(* IEC 61131-3 sources: Temperature-Cabinet-Control-Automation/src/POUs, 3 files *)

(* ---- FB_CabinetSetpointControl.st ---- *)
(*
    FUNCTION_BLOCK: FB_CabinetSetpointControl
    Project:  Temperature Cabinet Setpoint Control from CODESYS HMI
    Author:   OJ (Omkar Joshi) - Oliver Mechatronics
    Language: IEC 61131-3 Structured Text (CODESYS 3.5, WebVisu)

    ------------------------------------------------------------------
    ROLE
    Supervisory setpoint control for the Left Hand Small Temperature
    Cabinet (Watlow F4S, Modbus RTU / RS-232). CODESYS never runs the
    thermal loop - the F4S keeps its own closed-loop PID. This block:

      1. Takes a new desired setpoint from the HMI (GVL_HMI.rReqSetpoint).
      2. Validates it against safe limits.
      3. Writes it once (edge-triggered FC06) to register 300 (SP1).
      4. Confirms acceptance by reading register 300 back and comparing.
      5. Raises a clear, prioritised fault if the write fails, the link
         is lost, the value is refused, or the cabinet is over temperature.

    Matches the Project Development Package spec (Details A) and the
    build guide already in codesys-modbus-integration/README.md
    (Part 3, Part 4) and the T1-T9 test plan in the main README.

    SCALING
    F4S registers carry one implied decimal (raw 1300 == 130.0 degC).
    rScale defaults to 10.0; change it if the unit is reconfigured
    for a different resolution.

    NOTE (known follow-up item): this FB reads/writes GVL_Modbus and
    GVL_HMI directly in its body rather than exclusively through
    VAR_INPUT/VAR_OUTPUT. That is how the Project Development Package
    and the README build guide specify it, and it is what the T1-T9
    bench tests exercise - but it does mean this FB cannot be unit
    tested or reused against a second GVL_Modbus instance without
    editing the body. See PLC_PRG for the wired-up call, and note the
    xOverTempDI placeholder wiring there.
    ------------------------------------------------------------------
*)
FUNCTION_BLOCK FB_CabinetSetpointControl
VAR_INPUT
    rRequestedSetpoint  : REAL;                    (* deg C from HMI                    *)
    xSetCommand         : BOOL;                    (* HMI SET - rising edge applies      *)
    xReset              : BOOL;                    (* fault reset - rising edge clears   *)
    xOverTempDI         : BOOL;                    (* spare EL1409 DI, TRUE = over-temp  *)

    (* ---- configurable, default to confirmed values ---- *)
    rMinSetpoint        : REAL := -40.0;           (* Lower safe bound, degC              *)
    rMaxSetpoint        : REAL := 200.0;           (* Upper safe bound, degC              *)
    rScale              : REAL := 10.0;            (* eng <-> raw multiplier              *)
    rTolerance          : REAL := 0.1;             (* deg C read-back tolerance           *)
    tCommsTimeout       : TIME := T#3S;            (* watchdog                            *)
END_VAR
VAR_OUTPUT
    eState              : E_SetpointState;
    eFault              : E_FaultCode;
    xConfirmed          : BOOL;
    xFault              : BOOL;
    rActualTemp         : REAL;                    (* Live chamber temperature, degC      *)
    rConfirmedSetpoint  : REAL;                    (* Last accepted setpoint, degC        *)
END_VAR
VAR
    rtrigSet            : R_TRIG;                  (* Edge detect on SET command          *)
    rtrigReset          : R_TRIG;                  (* Edge detect on RESET command        *)
    tonWatchdog         : TON;                     (* Comms-loss debounce                 *)
    tonConfirmWait      : TON;                     (* Read-back confirm timeout           *)
    wTargetRaw          : WORD;                    (* Setpoint being written, raw x10     *)
    rReadBack           : REAL;                    (* Setpoint echo, engineering units    *)
END_VAR

(* ---- Edge detect ---- *)
rtrigSet(CLK := xSetCommand);
rtrigReset(CLK := xReset);

(* ---- Always-live scaling of the cyclic read ---- *)
rActualTemp          := WORD_TO_REAL(GVL_Modbus.wInput1Value) / rScale;
rReadBack             := WORD_TO_REAL(GVL_Modbus.wSetpoint1Read) / rScale;
GVL_HMI.rChamberTemp := rActualTemp;

(* ---- Comms watchdog: LEVEL signal, NOT an edge pulse (avoids R_TRIG->TON trap) ---- *)
tonWatchdog(IN := NOT GVL_Modbus.xModbusDone, PT := tCommsTimeout);

(* ---- Over-temp interlock (highest priority latch) ---- *)
IF xOverTempDI THEN
    eFault := E_FaultCode.OVER_TEMP;
    eState := E_SetpointState.FAULTED;
END_IF

(* ---- Comms loss latch (any state) ---- *)
IF tonWatchdog.Q OR GVL_Modbus.xModbusError THEN
    eFault := E_FaultCode.COMMS_TIMEOUT;
    eState := E_SetpointState.FAULTED;
END_IF

CASE eState OF

    E_SetpointState.IDLE:
        xConfirmed := TRUE;
        GVL_Modbus.xWriteTrigger := FALSE;
        IF rtrigSet.Q THEN
            eState := E_SetpointState.READY;
        END_IF

    E_SetpointState.READY:
        xConfirmed := FALSE;
        IF rRequestedSetpoint < rMinSetpoint THEN
            eFault := E_FaultCode.RANGE_LOW;
            eState := E_SetpointState.FAULTED;
        ELSIF rRequestedSetpoint > rMaxSetpoint THEN
            eFault := E_FaultCode.RANGE_HIGH;
            eState := E_SetpointState.FAULTED;
        ELSE
            wTargetRaw := REAL_TO_WORD(rRequestedSetpoint * rScale);
            GVL_Modbus.wSetpoint1Write := wTargetRaw;
            eState := E_SetpointState.WRITING;
        END_IF

    E_SetpointState.WRITING:
        GVL_Modbus.xWriteTrigger := TRUE;    (* one-shot rising edge fires FC06 *)
        eState := E_SetpointState.CONFIRM;

    E_SetpointState.CONFIRM:
        GVL_Modbus.xWriteTrigger := FALSE;   (* drop trigger to re-arm the edge *)
        tonConfirmWait(IN := TRUE, PT := tCommsTimeout);
        IF ABS(rReadBack - rRequestedSetpoint) <= rTolerance THEN
            rConfirmedSetpoint := rReadBack;
            GVL_HMI.rConfirmedSetpoint := rReadBack;
            tonConfirmWait(IN := FALSE);
            eState := E_SetpointState.IDLE;
        ELSIF tonConfirmWait.Q THEN
            eFault := E_FaultCode.NOT_ACCEPTED;
            eState := E_SetpointState.FAULTED;
        END_IF

    E_SetpointState.FAULTED:
        xConfirmed := FALSE;
        GVL_Modbus.xWriteTrigger := FALSE;
        (* Latched - clears only on reset edge AND only if condition is gone *)
        IF rtrigReset.Q
           AND NOT xOverTempDI
           AND NOT tonWatchdog.Q
           AND NOT GVL_Modbus.xModbusError THEN
            eFault := E_FaultCode.NO_FAULT;
            eState := E_SetpointState.IDLE;
        END_IF

END_CASE

xFault                      := (eState = E_SetpointState.FAULTED);
GVL_HMI.xSetpointConfirmed  := xConfirmed AND NOT xFault;
GVL_HMI.xFaultActive        := xFault;
GVL_HMI.eFaultCode          := eFault;

(* ---- PLC_PRG.st ---- *)
(*
    PROGRAM:  PLC_PRG
    Project:  Temperature Cabinet Setpoint Control from CODESYS HMI
    Author:   OJ (Omkar Joshi) - Oliver Mechatronics
    Language: IEC 61131-3 Structured Text (CODESYS 3.5, WebVisu)

    Cyclic entry point (MainTask). Instantiates the supervisory setpoint
    controller. Because FB_CabinetSetpointControl reads/writes GVL_Modbus
    and GVL_HMI directly in its body (see that FB's header note), this
    program only needs to pass through the operator-facing parameters
    and the safety interlock input.

    Matches the Project Development Package spec (Details A) and the
    build guide already in codesys-modbus-integration/README.md.

    TODO (flagged in the Project Development Package, not yet resolved):
    xOverTempDI below is wired to GVL_Modbus.xModbusError as a
    placeholder. REPLACE with the real mapped EL1409 digital-input
    channel (spare over-temperature lamp contact) in the EtherCAT I/O
    mapping before relying on this interlock.
*)
PROGRAM PLC_PRG
VAR
    fbSetpoint : FB_CabinetSetpointControl;
END_VAR

(* ---- Drive the supervisory setpoint controller ---- *)
fbSetpoint(
    rRequestedSetpoint := GVL_HMI.rReqSetpoint,
    xSetCommand        := GVL_HMI.xSetBtn,
    xReset             := GVL_HMI.xResetBtn,
    xOverTempDI        := GVL_Modbus.xModbusError,  (* REPLACE with mapped EL1409 DI channel *)
    rMinSetpoint       := 30.0,
    rMaxSetpoint       := 130.0
);

(* ---- Consume dialog button one-shots ---- *)
GVL_HMI.xSetBtn   := FALSE;
GVL_HMI.xResetBtn := FALSE;

(* ---- PLC_PRG_TCP_Retargeted.st ---- *)
PROGRAM PLC_PRG
(* ======================================================================
   Retargeted for TCP register sources (Python gateway via Modbus TCP)
   ======================================================================
   Serial device abandoned. All reads/writes now come via the TCP slave
   device on the Modbus TCP master branch of the device tree.

   Proven register map (TCP holding registers, x10 integers):
     reg2 = chamber temperature (read-only, cyclic)
     reg3 = confirmed setpoint read-back (read-only, cyclic)
     reg4 = status/fault code (read-only, cyclic)
     reg0 = requested setpoint (write, cyclic or rising)
     reg1 = apply trigger (write, rising edge)

   I/O Mapping binds these to GVL_Modbus:
     reg2 -> wInput1Value (temperature)
     reg3 -> wSetpoint1Read (confirmed SP)
     reg4 -> wStatus (fault code: 0=OK, 2=WRITE_FAILED, 3=NOT_ACCEPTED, 4=RANGE, 5=COMMS)
     reg0 -> wSetpoint1Write (requested SP, x10)
     reg1 -> xWriteTrigger (apply pulse, BOOL as WORD 0/1)

   The state machine logic is unchanged from the serial version. Only the
   data sources changed: TCP channels instead of serial channels.
   ====================================================================== *)

VAR
    rChamberTemp        : REAL;
    rReqSetpoint        : REAL := 26.5;           (* set in watch window or WebVisu *)
    rConfirmedSetpoint  : REAL;

    rMinSetpoint        : REAL := -40.0;
    rMaxSetpoint        : REAL := 200.0;

    eSetpointState      : E_SetpointState := E_SetpointState.IDLE;
    eFaultCode          : E_FaultCode := E_FaultCode.NO_FAULT;

    xStartWrite         : BOOL := FALSE;          (* rising-edge trigger for manual test *)
    xPrevStartWrite     : BOOL := FALSE;
    xWriteTriggered     : BOOL := FALSE;

    dwWriteTimeout      : DWORD := 0;
    dwMaxTimeout        : DWORD := 300;           (* ~3s at 10ms MainTask *)
END_VAR

(* --- STEP 1: Scale raw TCP values -> engineering units ---
   TCP registers carry x10 integers; we work in real degrees.
   All three reads come from the TCP channels (wInput1Value, wSetpoint1Read, wStatus).
*)
rChamberTemp       := GVL_Modbus.wInput1Value / 10.0;
rConfirmedSetpoint := GVL_Modbus.wSetpoint1Read / 10.0;

(* --- STEP 2: Detect rising edge on the manual test trigger ---
   When testing from watch window, toggle xStartWrite from FALSE to TRUE.
   In production (WebVisu or SCADA), the operator triggers via a button that
   sets a HMI variable, but the edge logic is the same.
*)
xWriteTriggered := (xStartWrite AND NOT xPrevStartWrite);
xPrevStartWrite := xStartWrite;

(* --- STEP 3: State machine (unchanged logic, TCP-based register sources) --- *)

CASE eSetpointState OF

    E_SetpointState.IDLE:
        (* Waiting for a write request. Hold the apply trigger low. *)
        GVL_Modbus.xWriteTrigger := FALSE;
        dwWriteTimeout := 0;

        IF xWriteTriggered THEN
            eSetpointState := E_SetpointState.READY;
        END_IF

    E_SetpointState.READY:
        (* Validate the requested setpoint against limits. *)
        IF rReqSetpoint < rMinSetpoint THEN
            eFaultCode := E_FaultCode.RANGE_LOW;
            eSetpointState := E_SetpointState.FAULTED;

        ELSIF rReqSetpoint > rMaxSetpoint THEN
            eFaultCode := E_FaultCode.RANGE_HIGH;
            eSetpointState := E_SetpointState.FAULTED;

        ELSE
            (* Valid range. Stage the request (x10 int) into the TCP write register. *)
            GVL_Modbus.wSetpoint1Write := DWORD_TO_WORD(REAL_TO_DWORD(rReqSetpoint * 10.0));
            eSetpointState := E_SetpointState.WRITING;
        END_IF

    E_SetpointState.WRITING:
        (* Pulse the apply trigger (one scan). The Python gateway services this
           by writing reg1=1 over RTU and then clearing it to 0 when done. *)
        GVL_Modbus.xWriteTrigger := TRUE;
        dwWriteTimeout := 0;
        eSetpointState := E_SetpointState.CONFIRM;

    E_SetpointState.CONFIRM:
        (* Drop the trigger immediately to re-arm the edge for the next request. *)
        GVL_Modbus.xWriteTrigger := FALSE;
        dwWriteTimeout := dwWriteTimeout + 1;

        (* Check for immediate comms failure (Python gateway lost). *)
        IF GVL_Modbus.wStatus = 5 THEN                  (* COMMS fault from gateway *)
            eFaultCode := E_FaultCode.COMMS_TIMEOUT;
            eSetpointState := E_SetpointState.FAULTED;

        (* Check for write-accepted confirmation: read-back matches request. *)
        ELSIF ABS(rConfirmedSetpoint - rReqSetpoint) < 0.1 THEN
            eFaultCode := E_FaultCode.NO_FAULT;
            eSetpointState := E_SetpointState.IDLE;

        (* Check for write-failed fault (Python couldn't write to F4S). *)
        ELSIF GVL_Modbus.wStatus = 2 THEN                (* WRITE_FAILED *)
            eFaultCode := E_FaultCode.WRITE_FAILED;
            eSetpointState := E_SetpointState.FAULTED;

        (* Check for not-accepted fault (F4S silent-rejected, e.g., menu mode). *)
        ELSIF GVL_Modbus.wStatus = 3 THEN                (* NOT_ACCEPTED *)
            eFaultCode := E_FaultCode.NOT_ACCEPTED;
            eSetpointState := E_SetpointState.FAULTED;

        (* Check for range/fault from Python side. *)
        ELSIF GVL_Modbus.wStatus = 4 THEN                (* RANGE *)
            eFaultCode := E_FaultCode.RANGE_HIGH;        (* or RANGE_LOW; Python validates *)
            eSetpointState := E_SetpointState.FAULTED;

        (* Timeout: Python didn't respond in time. *)
        ELSIF dwWriteTimeout > dwMaxTimeout THEN
            eFaultCode := E_FaultCode.NOT_ACCEPTED;      (* treated as F4S rejection *)
            eSetpointState := E_SetpointState.FAULTED;
        END_IF

    E_SetpointState.FAULTED:
        (* Latched fault state. User must acknowledge by re-triggering (watch window or HMI). *)
        GVL_Modbus.xWriteTrigger := FALSE;

        IF xWriteTriggered THEN
            eFaultCode := E_FaultCode.NO_FAULT;
            eSetpointState := E_SetpointState.READY;
        END_IF

END_CASE

(* --- STEP 4: Consume the manual test trigger (so it doesn't re-fire) ---
   In production, replace xStartWrite with the HMI/WebVisu button signal.
   The gateway's apply trigger (reg1) is cleared by the Python side after processing.
*)
xStartWrite := FALSE;
